// Mitsubishi GX Works2 project: team1   PLC: FX3G

// global labels: Global1
VAR_GLOBAL
  start_day AT X007 : BOOL;
  shmarim_count AT CC1 : BOOL;
  letet_count AT CC2 : BOOL;
  kshut_count AT CC3 : BOOL;
  analog_output AT D8282 : INT;
  total_packs AT D1100 : INT;
  input_shmarim AT D1110 : INT;
  shmarim_amount AT D1120 : INT;
  input_letet AT D1130 : INT;
  letet_amount AT D1140 : INT;
  input_kshut AT D1150 : INT;
  kshut_amount AT D1160 : INT;
  end_day AT X011 : BOOL;
  day_light AT Y007 : BOOL;
  M_10 AT M10 : BOOL;
  start_cooking AT X001 : BOOL;
  analog_input2 AT D8281 : REAL;
END_VAR
VAR_GLOBAL CONSTANT
  pilzner_lower_limit : INT := 6;
END_VAR
VAR_GLOBAL
  pilzner_selected AT M12 : BOOL;
END_VAR
VAR_GLOBAL CONSTANT
  lager_lower_limit : INT := 5;
END_VAR
VAR_GLOBAL
  lager_selected AT M13 : BOOL;
END_VAR
VAR_GLOBAL CONSTANT
  pilzner_shmarim_limit : INT := 120;
  pilzner_letet_limit : INT := 6;
  pilzner_kshut_limit : INT := 54;
END_VAR
VAR_GLOBAL
  pilzner_start AT M14 : BOOL;
  check_light AT TS1 : BOOL;
  light AT Y001 : BOOL;
  tc1 AT TC1 : BOOL;
END_VAR
VAR_GLOBAL CONSTANT
  timer_cook_light : INT := 40;
END_VAR
VAR_GLOBAL
  analog_input1 AT D8280 : INT;
  save_analog_value AT D7778 : INT;
END_VAR
VAR_GLOBAL CONSTANT
  divide_num : INT := 400;
  lager_shmarim_limit : INT := 150;
  lager_letet_limit : INT := 12;
  lager_kshut_limit : INT := 60;
END_VAR
VAR_GLOBAL
  lager_start AT M15 : BOOL;
  check AT Y002 : BOOL;
  start_fermentation AT X005 : BOOL;
  finish_cooking AT Y001 : BOOL;
  M_17 AT M17 : BOOL;
  M_0 AT M0 : BOOL;
  tc_2 AT TC2 : BOOL;
END_VAR
VAR_GLOBAL CONSTANT
  lager_fermentation_time : INT := 30;
END_VAR
VAR_GLOBAL
  ts_2 AT TS2 : BOOL;
  tc_3 AT TC3 : BOOL;
  ts_3 AT TS3 : BOOL;
  M_1 AT M1 : BOOL;
  ts_4 AT TS4 : BOOL;
  tc_4 AT TC4 : BOOL;
END_VAR
VAR_GLOBAL CONSTANT
  pilzner_fermentation_time : INT := 40;
END_VAR
VAR_GLOBAL
  tc_5 AT TC5 : BOOL;
  ts_5 AT TS5 : BOOL;
  M_23 AT M23 : BOOL;
  Y_3 AT Y003 : BOOL;
  Y_4 AT Y004 : BOOL;
END_VAR
VAR_GLOBAL CONSTANT
  blink_time : INT := 5;
END_VAR
VAR_GLOBAL
  packing_start AT X002 : BOOL;
  packing_one_bottle AT X000 : BOOL;
  bottles_counter AT CC6 : BOOL;
  M_25 AT M25 : BOOL;
  M_16 AT M16 : BOOL;
  one_bottle_packing AT X000 : BOOL;
  one_bottle_start AT CC4 : BOOL;
END_VAR
VAR_GLOBAL CONSTANT
  one_bottle_packed : INT := 1;
END_VAR
VAR_GLOBAL
  six_bottle_end AT CC5 : BOOL;
END_VAR
VAR_GLOBAL CONSTANT
  six_bottle_packed : INT := 6;
END_VAR
VAR_GLOBAL
  packing_end AT M11 : BOOL;
  first_bottle AT CS4 : BOOL;
  six_bottle AT CS5 : BOOL;
  packing_in_process AT Y002 : BOOL;
END_VAR
VAR_GLOBAL CONSTANT
  add_1 : INT := 1;
  reset_input1 : INT := 30;
  reset_input2 : INT := 50;
END_VAR
VAR_GLOBAL
  shmarim_pilzner_check AT M18 : BOOL;
  letet_pilzner_check AT M19 : BOOL;
  kshut_pilzner_check AT M20 : BOOL;
  shmarim_lager_check AT M21 : BOOL;
  letet_lager_check AT M22 : BOOL;
  kshut_lager_check AT M23 : BOOL;
END_VAR
VAR_GLOBAL CONSTANT
  Mul_num : INT := 40;
END_VAR
VAR_GLOBAL
  outpot_mul AT D1200 : INT;
  analog_light AT M24 : BOOL;
END_VAR

// task Task_01 (event TRUE, interval 0, priority 31): POU_01

PROGRAM POU_01
(* structured ladder/FBD written out as ST: instructions are called as NAME(EN, inputs, outputs); _pN, _eN, _tN stand for wires *)
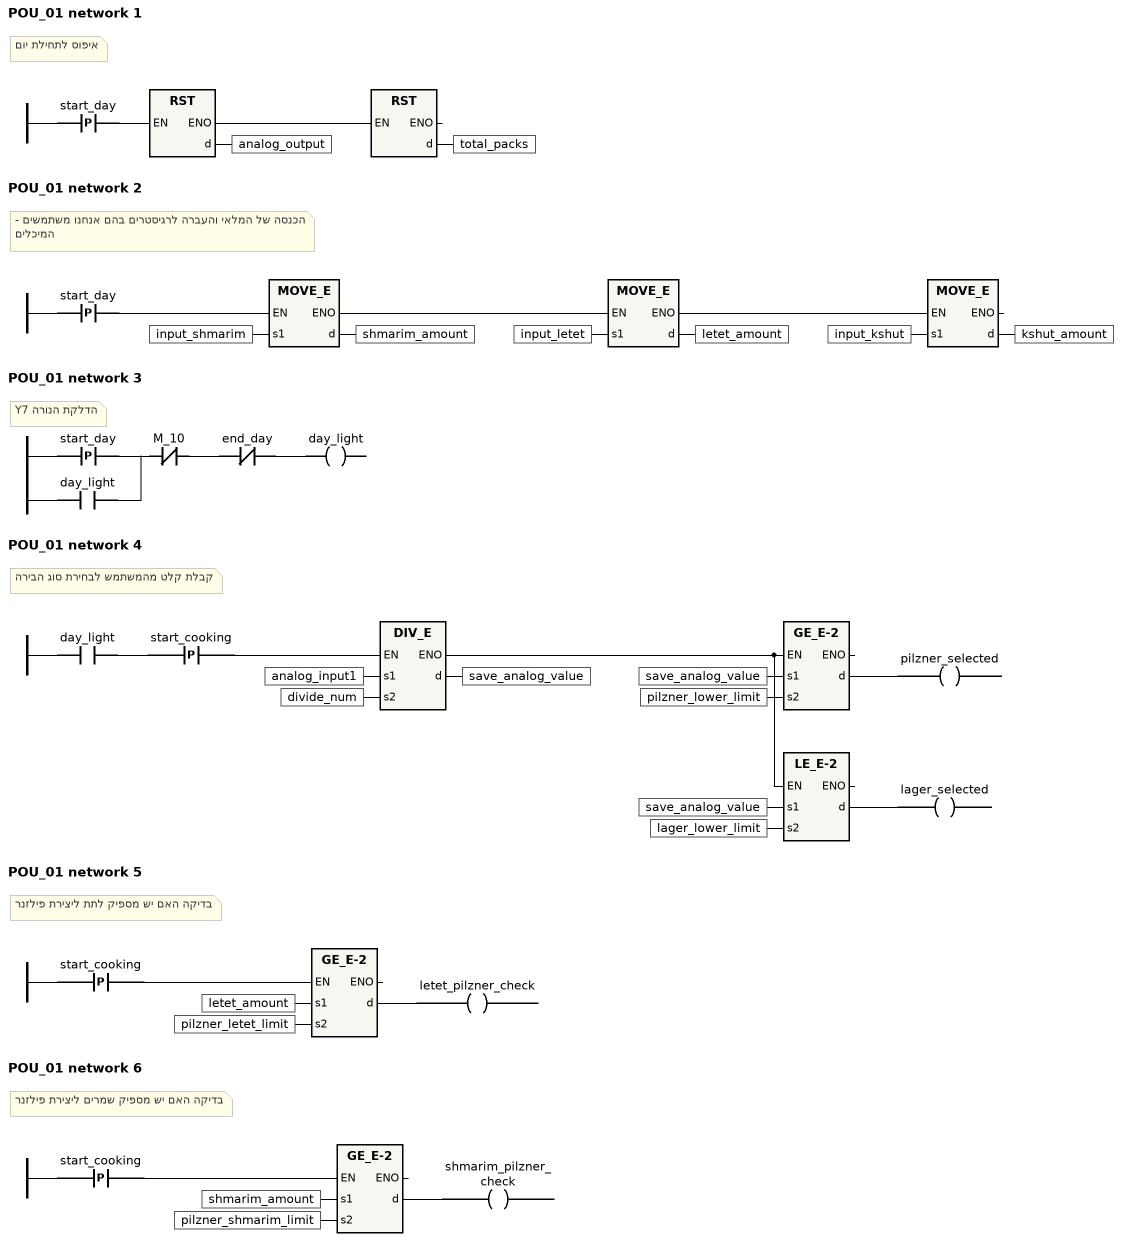
(* network 1 *)
(* איפוס לתחילת יום *)
_e1 := RST(LDP(TRUE, start_day), analog_output);
RST(_e1, total_packs);
(* network 2 *)
(* הכנסה של המלאי והעברה לרגיסטרים בהם אנחנו משתמשים - המיכלים *)
_e1 := MOVE_E(LDP(TRUE, start_day), input_shmarim, shmarim_amount);
_e2 := MOVE_E(_e1, input_letet, letet_amount);
MOVE_E(_e2, input_kshut, kshut_amount);
(* network 3 *)
(* הדלקת הנורה Y7 *)
day_light := ((LDP(TRUE, start_day) OR day_light) AND NOT M_10) AND NOT end_day;
(* network 4 *)
(* קבלת קלט מהמשתמש לבחירת סוג הבירה *)
_e1 := DIV_E(day_light AND LDP(TRUE, start_cooking), analog_input1, divide_num, save_analog_value);
GE_E(_e1, save_analog_value, pilzner_lower_limit, _t2);
pilzner_selected := _t2;
LE_E(_e1, save_analog_value, lager_lower_limit, _t3);
lager_selected := _t3;
(* network 5 *)
(* בדיקה האם יש מספיק לתת ליצירת פילזנר *)
GE_E(LDP(TRUE, start_cooking), letet_amount, pilzner_letet_limit, _t1);
letet_pilzner_check := _t1;
(* network 6 *)
(* בדיקה האם יש מספיק שמרים ליצירת פילזנר *)
GE_E(LDP(TRUE, start_cooking), shmarim_amount, pilzner_shmarim_limit, _t1);
shmarim_pilzner_check := _t1;
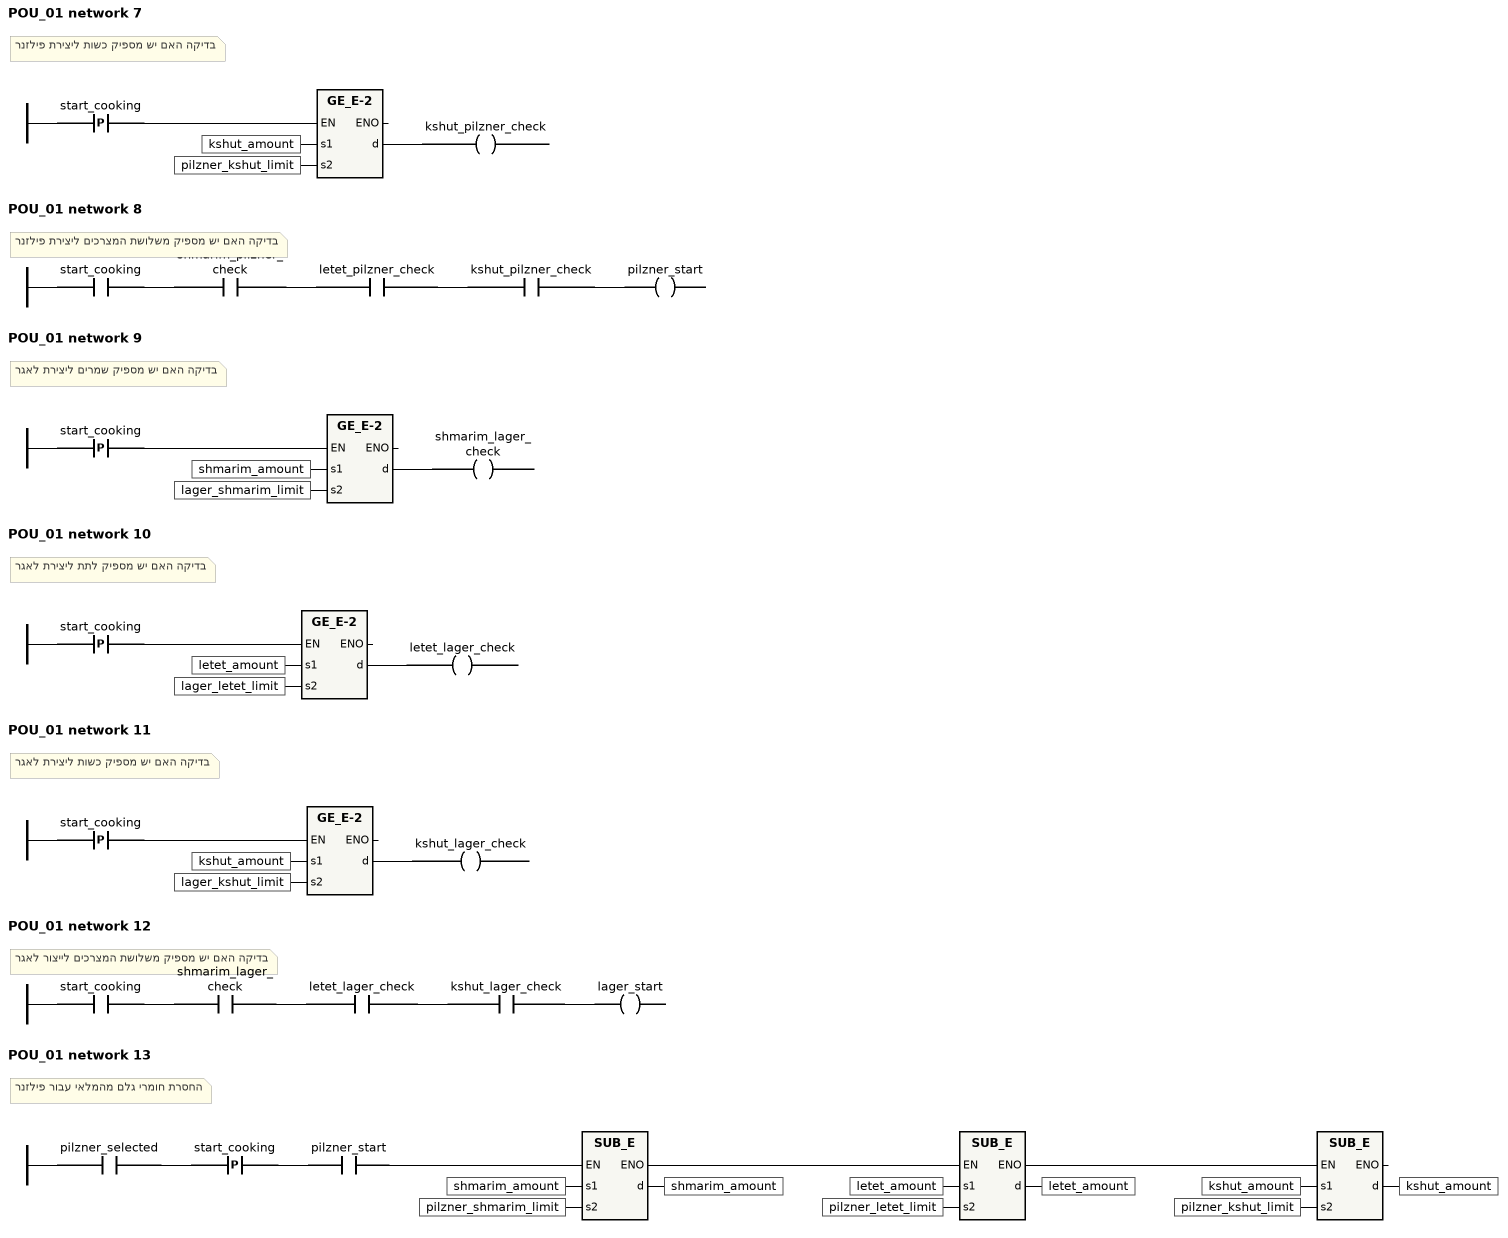
(* network 7 *)
(* בדיקה האם יש מספיק כשות ליצירת פילזנר *)
GE_E(LDP(TRUE, start_cooking), kshut_amount, pilzner_kshut_limit, _t1);
kshut_pilzner_check := _t1;
(* network 8 *)
(* בדיקה האם יש מספיק משלושת המצרכים ליצירת פילזנר *)
pilzner_start := start_cooking AND shmarim_pilzner_check AND letet_pilzner_check AND kshut_pilzner_check;
(* network 9 *)
(* בדיקה האם יש מספיק שמרים ליצירת לאגר *)
GE_E(LDP(TRUE, start_cooking), shmarim_amount, lager_shmarim_limit, _t1);
shmarim_lager_check := _t1;
(* network 10 *)
(* בדיקה האם יש מספיק לתת ליצירת לאגר *)
GE_E(LDP(TRUE, start_cooking), letet_amount, lager_letet_limit, _t1);
letet_lager_check := _t1;
(* network 11 *)
(* בדיקה האם יש מספיק כשות ליצירת לאגר *)
GE_E(LDP(TRUE, start_cooking), kshut_amount, lager_kshut_limit, _t1);
kshut_lager_check := _t1;
(* network 12 *)
(* בדיקה האם יש מספיק משלושת המצרכים לייצור לאגר *)
lager_start := start_cooking AND shmarim_lager_check AND letet_lager_check AND kshut_lager_check;
(* network 13 *)
(* החסרת חומרי גלם מהמלאי עבור פילזנר *)
_e1 := SUB_E(pilzner_selected AND LDP(TRUE, start_cooking) AND pilzner_start, shmarim_amount, pilzner_shmarim_limit, shmarim_amount);
_e2 := SUB_E(_e1, letet_amount, pilzner_letet_limit, letet_amount);
SUB_E(_e2, kshut_amount, pilzner_kshut_limit, kshut_amount);
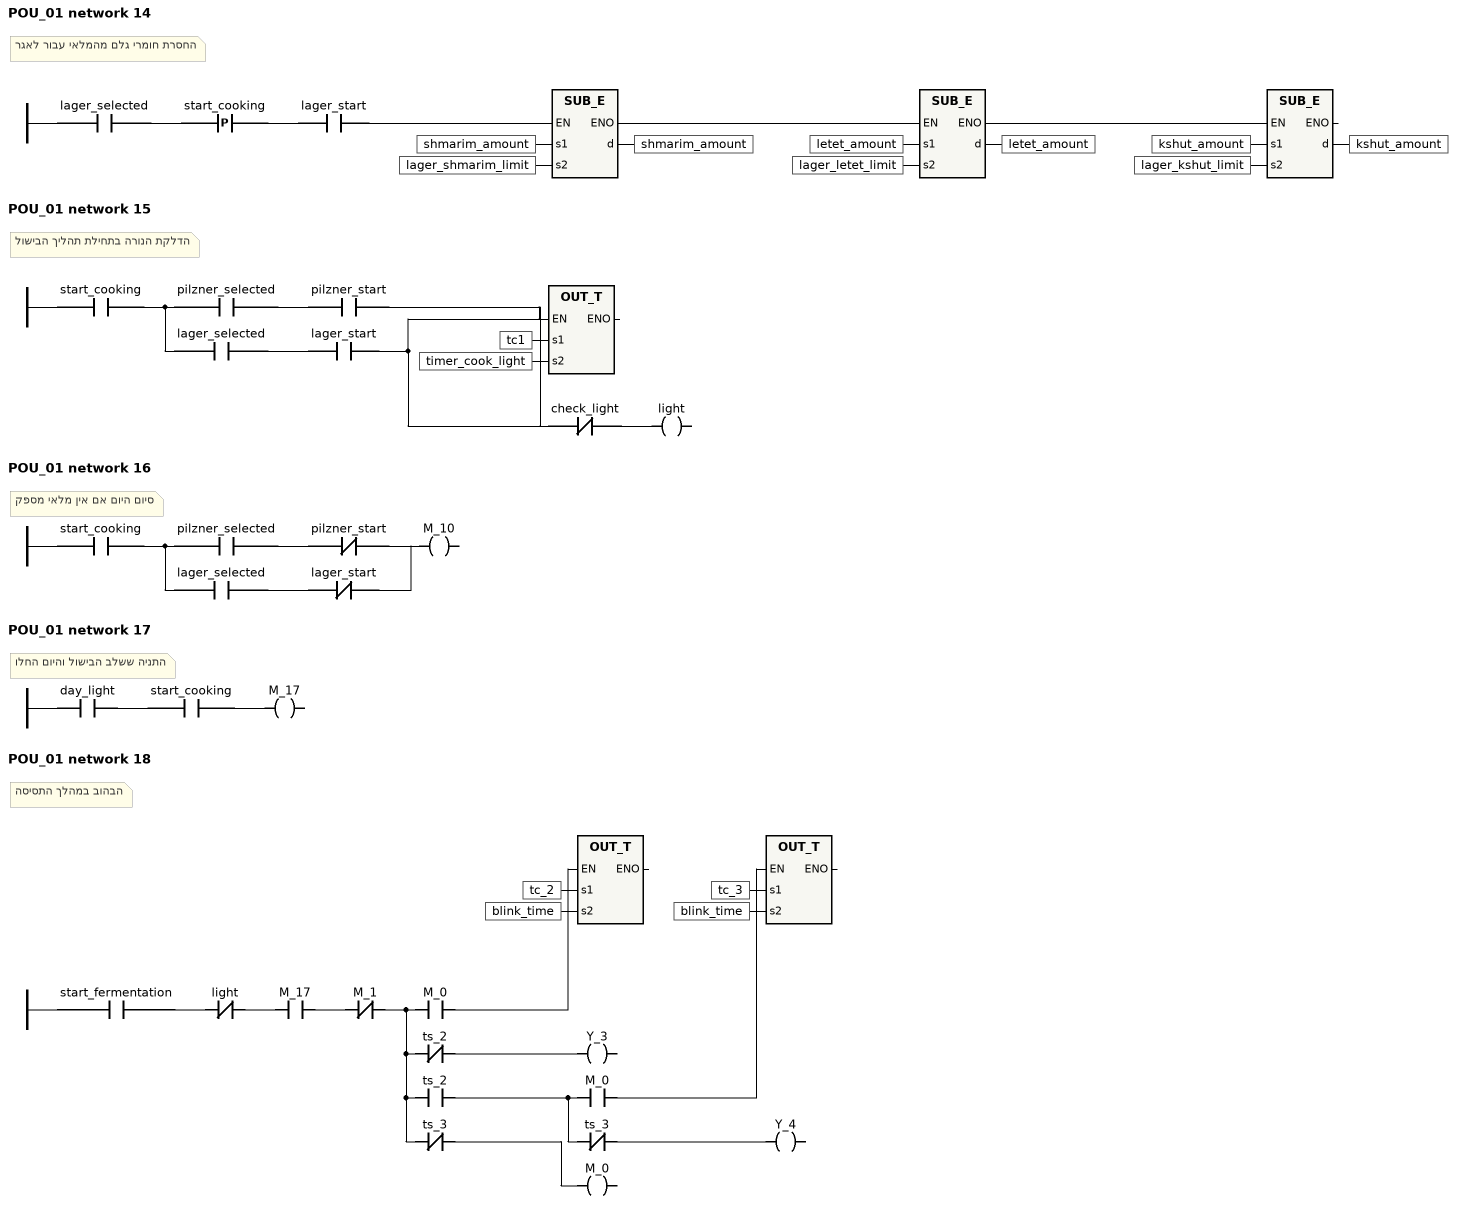
(* network 14 *)
(* החסרת חומרי גלם מהמלאי עבור לאגר *)
_e1 := SUB_E(lager_selected AND LDP(TRUE, start_cooking) AND lager_start, shmarim_amount, lager_shmarim_limit, shmarim_amount);
_e2 := SUB_E(_e1, letet_amount, lager_letet_limit, letet_amount);
SUB_E(_e2, kshut_amount, lager_kshut_limit, kshut_amount);
(* network 15 *)
(* הדלקת הנורה בתחילת תהליך הבישול *)
_p1 := (start_cooking AND pilzner_selected AND pilzner_start) OR (start_cooking AND lager_selected AND lager_start);
light := _p1 AND NOT check_light;
OUT_T(_p1, tc1, timer_cook_light);
(* network 16 *)
(* סיום היום אם אין מלאי מספק *)
M_10 := (start_cooking AND pilzner_selected AND NOT pilzner_start) OR (start_cooking AND lager_selected AND NOT lager_start);
(* network 17 *)
(* התניה ששלב הבישול והיום החלו *)
M_17 := day_light AND start_cooking;
(* network 18 *)
(* הבהוב במהלך התסיסה *)
_p1 := start_fermentation AND NOT light AND M_17 AND NOT M_1;
OUT_T(_p1 AND M_0, tc_2, blink_time);
Y_3 := _p1 AND NOT ts_2;
_p2 := _p1 AND ts_2;
OUT_T(_p2 AND M_0, tc_3, blink_time);
Y_4 := _p2 AND NOT ts_3;
M_0 := _p1 AND NOT ts_3;
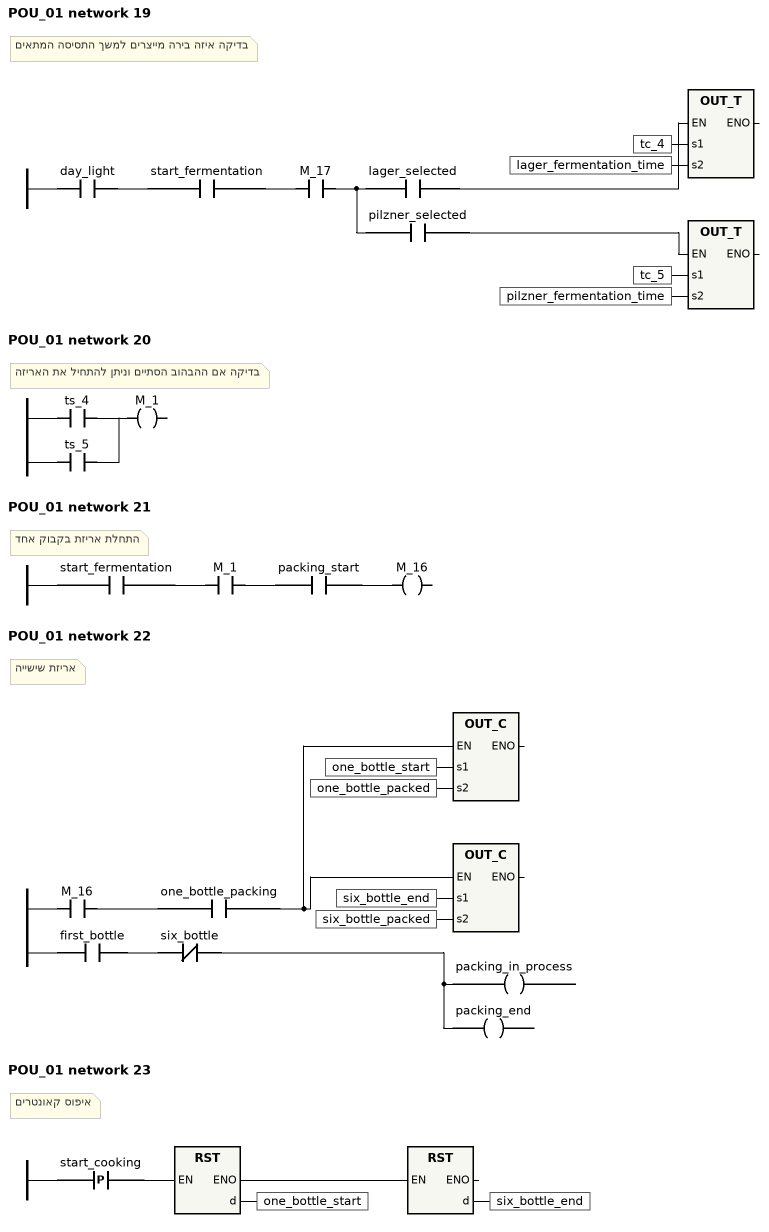
(* network 19 *)
(* בדיקה איזה בירה מייצרים למשך התסיסה המתאים *)
_p1 := day_light AND start_fermentation AND M_17;
OUT_T(_p1 AND lager_selected, tc_4, lager_fermentation_time);
OUT_T(_p1 AND pilzner_selected, tc_5, pilzner_fermentation_time);
(* network 20 *)
(* בדיקה אם ההבהוב הסתיים וניתן להתחיל את האריזה *)
M_1 := ts_4 OR ts_5;
(* network 21 *)
(* התחלת אריזת בקבוק אחד *)
M_16 := start_fermentation AND M_1 AND packing_start;
(* network 22 *)
(* אריזת שישייה *)
_p1 := M_16 AND one_bottle_packing;
OUT_C(_p1, one_bottle_start, one_bottle_packed);
OUT_C(_p1, six_bottle_end, six_bottle_packed);
_p2 := first_bottle AND NOT six_bottle;
packing_in_process := _p2;
packing_end := _p2;
(* network 23 *)
(* איפוס קאונטרים *)
_e1 := RST(LDP(TRUE, start_cooking), one_bottle_start);
RST(_e1, six_bottle_end);
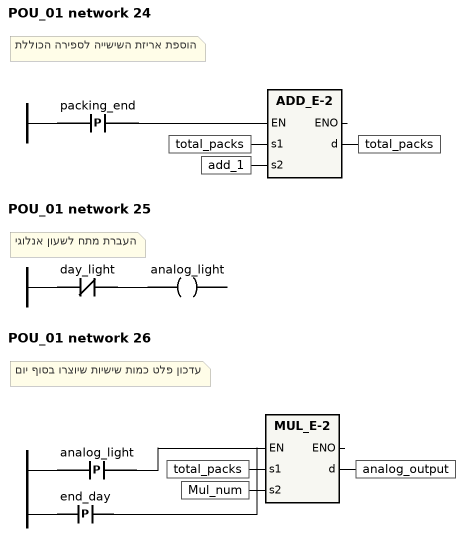
(* network 24 *)
(* הוספת אריזת השישייה לספירה הכוללת *)
ADD_E(LDP(TRUE, packing_end), total_packs, add_1, total_packs);
(* network 25 *)
(* העברת מתח לשעון אנלוגי *)
analog_light := NOT day_light;
(* network 26 *)
(* עדכון פלט כמות שישיות שיוצרו בסוף יום *)
MUL_E(LDP(TRUE, analog_light) OR LDP(TRUE, end_day), total_packs, Mul_num, analog_output);
END_PROGRAM
